(* CODESYS project raspberry_tcp_ip.project

Project tree, tasks and I/O mapping:
  Device : CODESYS Control for Raspberry Pi SL, 3S - Smart Software Solutions GmbH, version 3.5.12.10
    application Application
      libraries: Standard, * (System); Network, 3.5.7.0 (3S - Smart Software Solutions GmbH); BASIC, 3.3.3.0 (OSCAT); CAA DTUtil Extern, 3.5.12.0 (CAA Technical Workgroup); CAA Real Time Clock Extern, 3.5.10.0 (CAA Technical Workgroup); SysTime, 3.5.9.0 (System); CAA Mathematics, 3.5.12.0 (CAA Technical Workgroup)
      task MainTask (cyclic, interval 4 ms, priority 1) calls Update_Visu, TCP_Client
      task VISU_TASK (cyclic, interval 100 ms, priority 31) calls VisuElems.Visu_Prg
      program TCP_Client [ST]
      data type STATE
      visualisation Absolute_Movement
      global variables GVL
      visualisation Visualization
      function Math_Adjust [ST]
      program Update_Visu [ST]
      visualisation Relative_Movement
    Camera device
      <Empty>
    Onewire
    GPIOs_A_B : GPIOs A/B, 3S - Smart Software Solutions GmbH, version 3.5.11.0
        unmapped channels: digital inputs (GPIO0..GPIO31), digital outputs (GPIO0..GPIO31)
    SPI
    SoftMotion General Axis Pool
    I²C
  text list GlobalTextList
*)

// Device/Application/STATE
TYPE STATE :
(
	WAIT :=0,   (* Wait for on button to be pressed *)
	INIT, 	    (* Connections are set up and the message is created *)
	SEND,		(* Send message *)
	READ,		(* Receive and process message *)
	CANCEL,     (* Cancel the creation of a message *)
	ERROR		(* Prepare to reset connections *)
);
END_TYPE

// Device/Application/GVL
{attribute 'qualified_only'}
VAR_GLOBAL
	// 0 indicates absolute movement and 1 indicates relative movement
	mode: INT;
	home: BOOL;
	candle: BOOL;
	cancel: BOOL;
	ok: BOOL;
	on: BOOL;
	// 0 indicates radians and 1 indicates degrees
	anglesMode: BOOL;
	joint: ARRAY[1..6] OF REAL := [0.0, 0.87, 0.33, 0.0, 0.0, 0.0];
	initialPos: ARRAY[1..6] OF REAL;
	currentPos: ARRAY[1..6] OF STRING := ['0.0', '0.0', '0.0', '0.0', '0.0', '0.0'];
	error: ARRAY[1..6] OF REAL;
	desiredPos: ARRAY[1..6] OF REAL;
	poses: INT := 1;
END_VAR

// Device/Application/Update_Visu
// Program responsible to update visualization textfields, buttons etc. 
// regarding with the user's choices.
PROGRAM Update_Visu
VAR
	joint2MinStr: STRING;
	joint2MaxStr: STRING;
	joint3MinStr: STRING;
	joint3MaxStr: STRING;
	joint2Min: REAL;
	joint2Max: REAL;
	joint3Min: REAL;
	joint3Max: REAL;
	constraintsMin: ARRAY[1..6] OF REAL := [-3.14, 0.87, 0.33, -3.14, -3.14, -3.14];
	constraintsMax: ARRAY[1..6] OF REAL := [3.14, 5.41, 5.95, 3.14, 3.14, 3.14];
	anglesModeStr: STRING;
	jointVisu: ARRAY [1..6] OF STRING;
	errorVisu: ARRAY [1..6] OF STRING;
	currentPosVisu: ARRAY [1..6] OF STRING;
	constraintsMinVisu: ARRAY [1..6] OF STRING;
	constraintsMaxVisu: ARRAY [1..6] OF STRING;
	alarm: BOOL;
	alarm1: BOOL;
	alarm4: BOOL;
	alarm5: BOOL;
	alarm6: BOOL;
	i: INT;
END_VAR

// Update visualization elements according to user's choices
joint2Min:= OSCAT_BASIC.ROUND(constraintsMin[2] - GVL.initialPos[2], 2);
joint2Max:= OSCAT_BASIC.ROUND(constraintsMax[2] - GVL.initialPos[2], 2);
joint3Min:= OSCAT_BASIC.ROUND(constraintsMin[3] - GVL.initialPos[3], 2);
joint3Max:= OSCAT_BASIC.ROUND(constraintsMax[3] - GVL.initialPos[3], 2);

IF GVL.anglesMode = 0 THEN
	
	anglesModeStr:= 'DEG';
	
	FOR i:= 1 TO 6 DO
		jointVisu[i]:= REAL_TO_STRING(OSCAT_BASIC.ROUND(GVL.joint[i], 2));
		constraintsMinVisu[i]:= REAL_TO_STRING(constraintsMin[i]);
		constraintsMaxVisu[i]:= REAL_TO_STRING(constraintsMax[i]);
		currentPosVisu[i]:= REAL_TO_STRING(OSCAT_BASIC.ROUND(STRING_TO_REAL(GVL.currentPos[i]), 6));
		errorVisu[i]:= REAL_TO_STRING(OSCAT_BASIC.ROUND(GVL.error[i], 6));
	END_FOR
	
	joint2MinStr:= REAL_TO_STRING(joint2Min);
	joint2MaxStr:= REAL_TO_STRING(joint2Max);
	joint3MinStr:= REAL_TO_STRING(joint3Min);
	joint3MaxStr:= REAL_TO_STRING(joint3Max);
	
ELSIF GVL.anglesMode = 1 THEN
	
	anglesModeStr:= 'RAD';
	
	FOR i:= 1 TO 6 DO
		jointVisu[i]:= INT_TO_STRING(REAL_TO_INT(OSCAT_BASIC.ROUND(GVL.joint[i] / 3.14 * 180, 0)));
		constraintsMinVisu[i]:= INT_TO_STRING(REAL_TO_INT(OSCAT_BASIC.ROUND(constraintsMin[i] / 3.14 * 180, 0 )));
		constraintsMaxVisu[i]:= INT_TO_STRING(REAL_TO_INT(OSCAT_BASIC.ROUND(constraintsMax[i] / 3.14 * 180, 0)));
		currentPosVisu[i]:= INT_TO_STRING(REAL_TO_INT(OSCAT_BASIC.ROUND(STRING_TO_REAL(GVL.currentPos[i]) / 3.14 * 180, 2)));
		errorVisu[i]:= INT_TO_STRING(REAL_TO_INT(OSCAT_BASIC.ROUND(GVL.error[i] / 3.14 * 180, 2)));
	END_FOR
	
	joint2MinStr:= INT_TO_STRING(REAL_TO_INT(OSCAT_BASIC.ROUND(joint2Min / 3.14 * 180, 0)));
	joint2MaxStr:= INT_TO_STRING(REAL_TO_INT(OSCAT_BASIC.ROUND(joint2Max / 3.14 * 180, 0)));
	joint3MinStr:= INT_TO_STRING(REAL_TO_INT(OSCAT_BASIC.ROUND(joint3Min / 3.14 * 180, 0)));
	joint3MaxStr:= INT_TO_STRING(REAL_TO_INT(OSCAT_BASIC.ROUND(joint3max / 3.14 * 180, 0)));
		
END_IF

// Check if joints 1, 4, 5, 6 are about to reach 10000 degrees or -10000 degrees
IF STRING_TO_REAL(GVL.currentPos[1]) / 3.14 * 180 >= 9280 OR STRING_TO_REAL(GVL.currentPos[1]) / 3.14 * 180 <= -9280 THEN
	alarm1:= 1;
	alarm:= 1;
ELSIF STRING_TO_REAL(GVL.currentPos[4]) / 3.14 * 180 >= 9280 OR STRING_TO_REAL(GVL.currentPos[4]) / 3.14 * 180 <= -9280 THEN
	alarm4:= 1;
	alarm:= 1;
ELSIF STRING_TO_REAL(GVL.currentPos[5]) / 3.14 * 180 >= 9280 OR STRING_TO_REAL(GVL.currentPos[5]) / 3.14 * 180 <= -9280 THEN
	alarm5:= 1;
	alarm:= 1;
ELSIF STRING_TO_REAL(GVL.currentPos[6]) / 3.14 * 180 >= 9280 OR STRING_TO_REAL(GVL.currentPos[6]) / 3.14 * 180 <= -9280 THEN
	alarm6:= 1;
	alarm:= 1;
ELSE
	alarm1:= 0;
	alarm4:= 0;
	alarm5:= 0;
	alarm6:= 0;
	alarm:= 0;
END_IF

END_PROGRAM

// Device/Application/TCP_Client
// Program responsible to set up a connection with the server, send the
// appropriate angular position message to the server and receive their
// response. 
PROGRAM TCP_Client

VAR
	eSTATE			: STATE; (* State of the program *)
	
	IPAddress		: NBS.IP_ADDR; (* Server's IP Address *)
	uiPort			: UINT; (* Port No. *)
	// Received message
	sReceived: STRING;
	sToSend			: STRING; (* Transmitted message *)
	ctErrorCounter	: CAA.COUNT; (* Number of connection errors *)

	TCPClient		: NBS.TCP_Client; (* FB TCP Client *)
	TCPWrite		: NBS.TCP_Write; (* FB TCP Writer *)
	TCPRead			: NBS.TCP_Read; (* FB TCP Read *)
	
	TCPConnection	: CAA.HANDLE; (* Handle to the established connection *)
	
	// Helper variable
	xSend			: BOOL;
	// Helper variable
	xEnable			: BOOL;
	i: INT;
	firstPos: INT;
	lastPos: INT;
	length: INT;
	posNew: INT;
	posOld: INT;
	sReceivedNew: STRING;
END_VAR

CASE eSTATE OF
	
STATE.WAIT: // wait for button on to be pressed
	IF GVL.on THEN 
		eSTATE:= STATE.INIT;
	END_IF


STATE.INIT:  // establish connection to TCP server
	IPAddress.sAddr:= '155.207.33.165';
	uiPort:= 8080;
	xEnable:= TRUE;
	
	(* Client establishes a connection to a TCP Server on 155.207.33.165:8080 when start is selected*)
	TCPClient(xEnable:= xEnable, udiTimeOut:= 0, ipAddr:= IPAddress, uiPort:= uiPort, hConnection=> TCPConnection);
	
	sToSend:= '';  // empty message

	IF NOT(GVL.home) AND NOT(GVL.candle) THEN
		IF GVL.mode = 1 THEN
			sToSend:= INSERT(sToSend, '1 ', LEN(sToSend)); // 1 indicates relative movement
		ELSIF GVL.mode = 0 THEN  
			sToSend:= INSERT(sToSend, '0 ', LEN(sToSend)); // 0 indicates absolute movement
		END_IF
	
		FOR i:= 1 TO 6 DO	
			GVL.joint[i]:= OSCAT_BASIC.ROUND(GVL.joint[i], 2);
			sToSend:= INSERT(sToSend, CONCAT(REAL_TO_STRING(GVL.joint[i]),' '), LEN(sToSend)); // position defined by the user
		END_FOR
	ELSIF GVL.home THEN
		sToSend:= '0 0.0 2.9 1.3 4.2 1.4 0.0'; // home position - first 0 indicates absolute movement
	ELSIF GVL.candle THEN 
		sToSend:= '0 3.14 3.14 3.14 3.14 3.14 3.14'; // candle position - first 0 indicates absolute movement
	END_IF

	IF GVL.cancel THEN
		eSTATE:= STATE.CANCEL; // recreate the message if button cancel is pressed
	ELSIF GVL.ok THEN
		IF TCPClient.xActive THEN 
			eSTATE:= STATE.SEND;  // send message to server if button on is pressed
		ELSIF TCPClient.xError THEN
			eSTATE:= STATE.ERROR;
		END_IF
	END_IF
	
	
STATE.SEND:  // send created message
	IF TCPClient.xActive THEN
		xSend:= TRUE;
		TCPWrite(xExecute:= xSend, udiTimeOut:= 0, hConnection:= TCPConnection, szSize:= SIZEOF(sToSend), pData:= ADR(sToSend));	
		IF TCPWrite.xDone THEN
			GVL.ok:= 0;			
			TCPWrite(xExecute:= FALSE);	
			xSend:= FALSE;	
			
			eSTATE:= STATE.READ;			
		ELSIF TCPWrite.xError THEN
			eState:= STATE.ERROR;
		END_IF
	ELSE
		eSTATE:= STATE.ERROR;
	END_IF

	
STATE.READ:  // receive messages from server
	IF TCPClient.xActive AND TCPConnection <> CAA.gc_hINVALID THEN
		TCPRead(xEnable:= TRUE, hConnection:= TCPConnection, szSize:= SIZEOF(sReceived), pData:= ADR(sReceived));
		
		IF TCPRead.xReady THEN	
			// Retrieve current joint position from received message
			firstPos:= 1;
			lastPos:= 0;
			length:= 0;
			sReceivedNew:= TCP_Client.sReceived;
		
			FOR i:= 1 TO 5 DO
				lastPos:= FIND(sReceivedNew, ' ');
				length:= lastPos - firstPos;
				GVL.currentPos[i]:= MID(sReceivedNew, length, firstPos);		
				sReceivedNew:= MID(sReceivedNew, LEN(sReceivedNew) - lastPos, lastPos + 1);
			END_FOR
			GVL.currentPos[6]:= sReceivedNew;

			// Compute desired joint position	
			IF GVL.home THEN
				GVL.desiredPos[1]:= 0.0;
				GVL.desiredPos[2]:= 2.9;
				GVL.desiredPos[3]:= 1.3;
				GVL.desiredPos[4]:= 4.2;
				GVL.desiredPos[5]:= 1.4;
				GVL.desiredPos[6]:= 0.0;
				GVL.home:= 0;
			ELSIF GVL.candle THEN 
				FOR i:= 1 TO 6 DO
					GVL.desiredPos[i]:= 3.14;
				END_FOR
				GVL.candle:= 0;
			ELSE
				FOR i:= 1 TO 6 DO
					GVL.desiredPos[i]:= GVL.initialPos[i] + GVL.joint[i];
				END_FOR
			END_IF

			// Compute position error
			FOR i:= 1 TO 6 DO
				GVL.error[i]:= Math_Adjust(Math_Adjust(GVL.desiredPos[i]) - Math_Adjust(STRING_TO_REAL(GVL.currentPos[i])));
				GVL.error[i]:= OSCAT_BASIC.ROUND(in:= GVL.error[i], N:= 6);
			END_FOR

			// Set initial joint position for the next execution 
			FOR i:= 1 TO 6 DO
				GVL.initialPos[i]:= OSCAT_BASIC.ROUND(in:= STRING_TO_REAL(GVL.currentPos[i]), N:= 6);
			END_FOR
			
			eSTATE:= STATE.INIT;
			GVL.poses:= GVL.poses + 1;
			
		ELSIF TCPRead.xError THEN
			eState:= STATE.ERROR;
		END_IF
	ELSE
		eSTATE:= STATE.ERROR;
	END_IF
	
	
STATE.CANCEL:
	GVL.home:= 0;
	GVL.candle:= 0;
	GVL.cancel:= 0;
	eSTATE:= STATE.INIT;
	
	
STATE.ERROR:  // if there is an error, establish connection from start 
	ctErrorCounter:= ctErrorCounter + 1;
	xEnable := FALSE;
	eState := STATE.INIT;

END_CASE

END_PROGRAM

// Device/Application/Math_Adjust
// Function that computes the angular position error of each joint within the
// range of 0 to 2pi rad.
FUNCTION Math_Adjust : REAL
VAR_INPUT
	value: REAL;
END_VAR

IF value <= -3.14 OR value > 3.14 THEN
	Math_adjust:= LREAL_TO_REAL(MATH.fmod(lrX:= value, lrM:= 6.28));
	IF value <= -3.14 THEN 
		Math_adjust:= value + 6.28;
	ELSIF value > 3.14 THEN
		Math_adjust:= value - 6.28;
	END_IF
ELSE
	Math_adjust:= value;
END_IF

END_FUNCTION

// Device/Application/Absolute_Movement
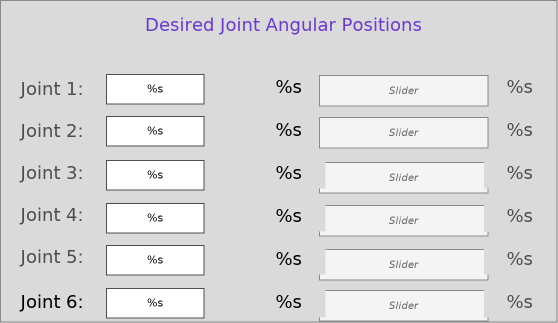
VISUALIZATION Absolute_Movement  // 558x323
    Slider (319,162 169x31), variable: GVL.joint[3], scale 0.33..5.95
    Slider (319,205 169x31), variable: GVL.joint[4], scale -3.14..3.14
    Slider (319,249 169x31), variable: GVL.joint[5], scale -3.14..3.14
    Slider (319,290 169x31), variable: GVL.joint[6], scale -3.14..3.14
    Label (111,10 345x30), "Desired Joint Angular Positions"
    Textfield (106,74 98x30), "%s", text variable: Update_Visu.jointVisu[1]
        OnMouseClick: write GVL.joint[1] via Edit
    Textfield (106,116 98x30), "%s", text variable: Update_Visu.jointVisu[2]
        OnMouseClick: write GVL.joint[2] via Edit
    Textfield (106,160 98x30), "%s", text variable: Update_Visu.jointVisu[3]
        OnMouseClick: write GVL.joint[3] via Edit
    Textfield (106,203 98x30), "%s", text variable: Update_Visu.jointVisu[4]
        OnMouseClick: write GVL.joint[4] via Edit
    Textfield (106,245 98x30), "%s", text variable: Update_Visu.jointVisu[5]
        OnMouseClick: write GVL.joint[5] via Edit
    Textfield (106,288 98x30), "%s", text variable: Update_Visu.jointVisu[6]
        OnMouseClick: write GVL.joint[6] via Edit
    Label (14,70 76x38), "Joint 1:"
    Label (14,112 76x38), "Joint 2:"
    Label (14,154 76x38), "Joint 3:"
    Label (14,196 76x38), "Joint 4:"
    Label (14,238 76x38), "Joint 5:"
    Label (14,283 76x38), "Joint 6:"
    Textfield (484,72 72x30), "%s", text variable: Update_Visu.constraintsMaxVisu[1]
    Textfield (484,115 72x30), "%s", text variable: Update_Visu.constraintsMaxVisu[2]
    Textfield (484,158 72x30), "%s", text variable: Update_Visu.constraintsMaxVisu[3]
    Textfield (484,201 72x30), "%s", text variable: Update_Visu.constraintsMaxVisu[4]
    Textfield (484,244 72x30), "%s", text variable: Update_Visu.constraintsMaxVisu[5]
    Textfield (484,287 72x30), "%s", text variable: Update_Visu.constraintsMaxVisu[6]
    Textfield (253,72 72x30), "%s", text variable: Update_Visu.constraintsMinVisu[1]
    Textfield (253,115 72x30), "%s", text variable: Update_Visu.constraintsMinVisu[2]
    Textfield (253,158 72x30), "%s", text variable: Update_Visu.constraintsMinVisu[3]
    Textfield (253,201 72x30), "%s", text variable: Update_Visu.constraintsMinVisu[4]
    Textfield (253,244 72x30), "%s", text variable: Update_Visu.constraintsMinVisu[5]
    Textfield (253,287 72x30), "%s", text variable: Update_Visu.constraintsMinVisu[6]
    Slider (319,75 169x31), variable: GVL.joint[1], scale -3.14..3.14
    Slider (319,117 169x31), variable: GVL.joint[2], scale 0.87..5.41
END_VISUALIZATION

// Device/Application/Visualization
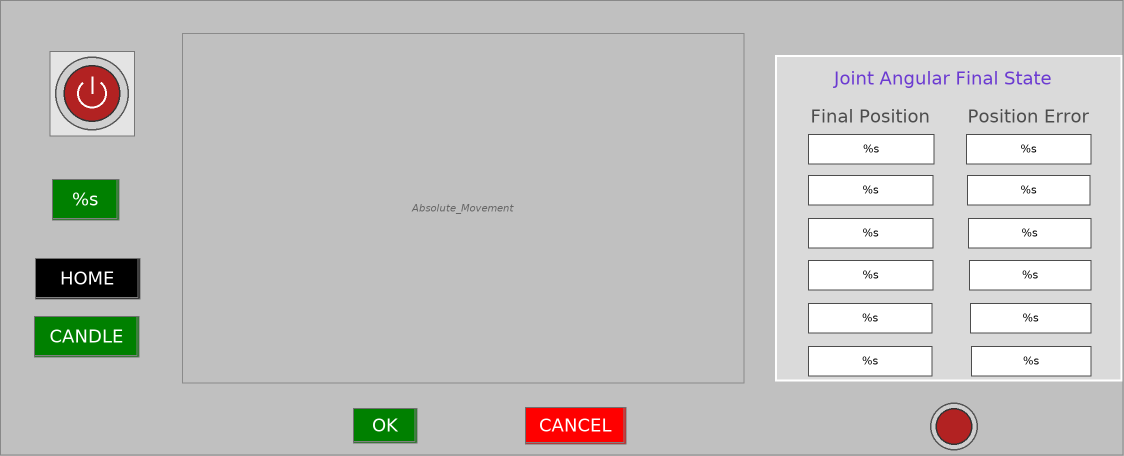
VISUALIZATION Visualization  // 1124x456
    Rectangle (775,55 347x326)
    PowerSwitch (47,51 90x85), variable: GVL.on, behaviour: TOGGLE, style: Switch-PowerSwitch-Red
    Textfield (808,134 126x30), "%s", text variable: Update_Visu.currentPosVisu[1], colour toggle: Update_Visu.alarm1
        p2167032090: 16#FF0000
    Textfield (808,175 125x30), "%s", text variable: Update_Visu.currentPosVisu[2]
    Textfield (808,218 125x30), "%s", text variable: Update_Visu.currentPosVisu[3]
    Textfield (808,260 125x30), "%s", text variable: Update_Visu.currentPosVisu[4], colour toggle: Update_Visu.alarm4
        p3092690914: 16#FF0000
    Textfield (808,303 124x30), "%s", text variable: Update_Visu.currentPosVisu[5], colour toggle: Update_Visu.alarm5
        p3092690914: 16#FF0000
    Textfield (808,346 124x30), "%s", text variable: Update_Visu.currentPosVisu[6], colour toggle: Update_Visu.alarm6
        p3092690914: 16#FF0000
    Label (800,100 141x33), "Final Position"
    TabControl (182,33 562x350), input disabled if: not (GVL.on), frame switch variable: GVL.mode
        shows Absolute_Movement()
        shows Relative_Movement()
        [0]: TabTitle=Absolute Movement
        [1]: TabTitle=Relative Movement
    Button (35,258 105x41), "HOME", input disabled if: not (GVL.on)
        toggle GVL.home
    Button (34,316 105x41), "CANDLE", input disabled if: not (GVL.on)
        toggle GVL.candle
    Label (797,66 292x25), "Joint Angular Final State"
    Textfield (966,134 125x30), "%s", text variable: Update_Visu.errorVisu[1]
    Textfield (967,175 123x30), "%s", text variable: Update_Visu.errorVisu[2]
    Textfield (968,218 123x30), "%s", text variable: Update_Visu.errorVisu[3]
    Textfield (969,260 122x30), "%s", text variable: Update_Visu.errorVisu[4]
    Textfield (970,303 121x30), "%s", text variable: Update_Visu.errorVisu[5]
    Textfield (971,346 120x30), "%s", text variable: Update_Visu.errorVisu[6]
    Label (959,100 139x33), "Position Error"
    Button (353,408 64x35), "OK", input disabled if: not (GVL.on)
        toggle GVL.ok
    Button (525,407 101x37), "CANCEL", input disabled if: not (GVL.on)
        toggle GVL.cancel
    Button (52,179 67x41), "%s", text variable: Update_Visu.anglesModeStr, input disabled if: not (GVL.on)
        toggle GVL.anglesMode
    Lamp1 (926,399 56x55), variable: Update_Visu.alarm, style: Lamp-Lamp1-Red
END_VISUALIZATION

// Device/Application/Relative_Movement
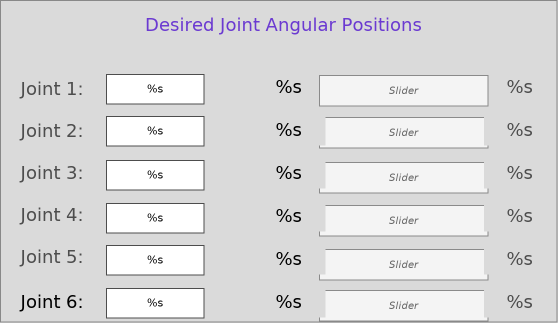
VISUALIZATION Relative_Movement  // 558x323
    Slider (319,117 169x31), variable: GVL.joint[2], scale 0.87..5.41
    Slider (319,162 169x31), variable: GVL.joint[3], scale 0.33..5.95
    Slider (319,205 169x31), variable: GVL.joint[4], scale -3.14..3.14
    Slider (319,249 169x31), variable: GVL.joint[5], scale -3.14..3.14
    Slider (319,290 169x31), variable: GVL.joint[6], scale -3.14..3.14
    Label (111,10 345x30), "Desired Joint Angular Positions"
    Textfield (106,74 98x30), "%s", text variable: Update_Visu.jointVisu[1]
        OnMouseClick: write GVL.joint[1] via Edit
    Textfield (106,116 98x30), "%s", text variable: Update_Visu.jointVisu[2]
        OnMouseClick: write GVL.joint[2] via Edit
    Textfield (106,160 98x30), "%s", text variable: Update_Visu.jointVisu[3]
        OnMouseClick: write GVL.joint[3] via Edit
    Textfield (106,203 98x30), "%s", text variable: Update_Visu.jointVisu[4]
        OnMouseClick: write GVL.joint[4] via Edit
    Textfield (106,245 98x30), "%s", text variable: Update_Visu.jointVisu[5]
        OnMouseClick: write GVL.joint[5] via Edit
    Textfield (106,288 98x30), "%s", text variable: Update_Visu.jointVisu[6]
        OnMouseClick: write GVL.joint[6] via Edit
    Label (14,70 76x38), "Joint 1:"
    Label (14,112 76x38), "Joint 2:"
    Label (14,154 76x38), "Joint 3:"
    Label (14,196 76x38), "Joint 4:"
    Label (14,238 76x38), "Joint 5:"
    Label (14,283 76x38), "Joint 6:"
    Textfield (484,72 72x30), "%s", text variable: Update_Visu.constraintsMaxVisu[1]
    Textfield (484,115 72x30), "%s", text variable: Update_Visu.joint2MaxStr
    Textfield (484,158 72x30), "%s", text variable: Update_Visu.joint3MaxStr
    Textfield (484,201 72x30), "%s", text variable: Update_Visu.constraintsMaxVisu[4]
    Textfield (484,244 72x30), "%s", text variable: Update_Visu.constraintsMaxVisu[5]
    Textfield (484,287 72x30), "%s", text variable: Update_Visu.constraintsMaxVisu[6]
    Textfield (253,72 72x30), "%s", text variable: Update_Visu.constraintsMinVisu[1]
    Textfield (253,115 72x30), "%s", text variable: Update_Visu.joint2MinStr
    Textfield (253,158 72x30), "%s", text variable: Update_Visu.joint3MinStr
    Textfield (253,201 72x30), "%s", text variable: Update_Visu.constraintsMinVisu[4]
    Textfield (253,244 72x30), "%s", text variable: Update_Visu.constraintsMinVisu[5]
    Textfield (253,287 72x30), "%s", text variable: Update_Visu.constraintsMinVisu[6]
    Slider (319,75 169x31), variable: GVL.joint[1], scale -3.14..3.14
END_VISUALIZATION
